// TIA Portal V19 export
TYPE "LubrValve_Pers"
// stored: Access Published
   STRUCT
      Par : "LubrValve_Par";
      ValvePumpCounter : Int;
      LubrReqCounter : LReal;
   END_STRUCT;
END_TYPE
